{attribute 'qualified_only'}
{attribute 'strict'}
{attribute 'to_string'}
TYPE E_State :
(
    Off,
    Init,
    Ready,
    Production,
    Done,
    Error,
    Stop,
    Setup
);
END_TYPE

(* stored: Version 1.1.0.1
   DUT E_State: Id {28e515e7-f34b-40d0-8c23-78f6a6a5ac15} *)
